// SIMATIC S7-200 project (STEP 7-Micro/WIN), CPU 221 REL 01.10

SYMBOL_TABLE USER1
start            I0.0     // khoi dong he thong
CB               I0.1     // cam bien
Y1               Q0.2     // di vao
Y2               Q0.1     // di ra
END_SYMBOL_TABLE

ORGANIZATION_BLOCK MAIN:OB1
TITLE=PROGRAM COMMENTS
BEGIN
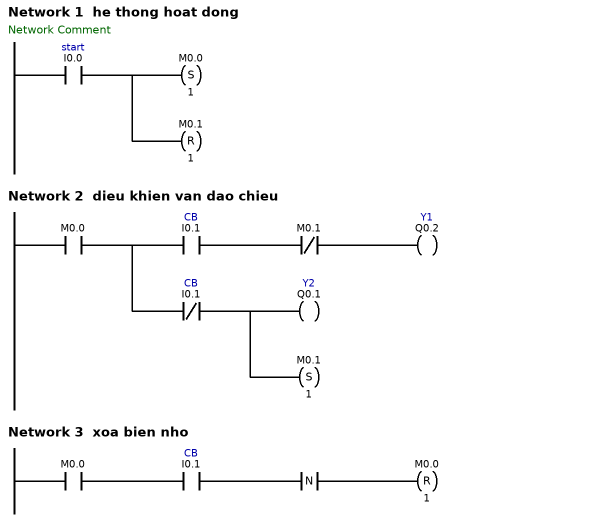
Network 1 // he thong hoat dong
// Network Comment
LD     start:I0.0
S      M0.0, 1
R      M0.1, 1
Network 2 // dieu khien van dao chieu
LD     M0.0
LPS
A      CB:I0.1
AN     M0.1
=      Y1:Q0.2
LPP
AN     CB:I0.1
=      Y2:Q0.1
S      M0.1, 1
Network 3 // xoa bien nho
LD     M0.0
A      CB:I0.1
ED
R      M0.0, 1
END_ORGANIZATION_BLOCK
